{attribute addProperty BoxType "EL5151-0080-0016"}
{attribute addProperty Id "ENC_InputsAT %I*ENC_Inputs_6FCA64CB112140ENC_Inputs_1AT %I*ENC_Inputs_AC51B8A03240ENC_OutputsAT %Q*ENC_Outputs_ADEB38374860WcStateAT %I*WcState_98A4DF7520.250InfoDataAT %I*InfoData_BC63D37F80100"}
{attribute addProperty CRC "1151073769"}
{attribute addProperty SizeInBites "274"}
{attribute addProperty SizeInBytes "34.25"}
TYPE EL5151_09E56EF0 :
STRUCT
	{attribute addProperty Name "ENC_Inputs"}
	ENC_Inputs : ENC_Inputs_6FCA64CB;
	{attribute addProperty Name "ENC_Inputs_1"}
	ENC_Inputs_1 : ENC_Inputs_AC51B8A0;
	{attribute addProperty Name "ENC_Outputs"}
	ENC_Outputs : ENC_Outputs_ADEB3837;
	{attribute addProperty Name "WcState"}
	WcState : WcState_98A4DF75;
	{attribute addProperty Name "InfoData"}
	InfoData : InfoData_BC63D37F;
END_STRUCT
END_TYPE

(* stored: Version 1.2.0.0, ProductVersion 3.1.4024.9
   DUT EL5151_09E56EF0: Id {14d0b1f3-9d4c-4e67-afe2-9a32c650b333} *)
